// TIA Portal V19 export
DATA_BLOCK "DecoilersHRot"   // DB66
// stored: InstanceOfName DecoilersHRot_FB, InstanceOfType FB
"DecoilersHRot_FB"
   // VAR_INPUT
   //    AreaInterface : "AreaInterface";
   //    ZSI : "udt_ZoneSafetyInterface";
   //    DSI : Struct
   //       Rotation : "udt_DeviceSafetyInterface";
   //       Pivot : "udt_DeviceSafetyInterface";
   //       Translation : "udt_DeviceSafetyInterface";
   //    END_STRUCT;
   //    Drive : Struct
   //       Traslation : "TAx_DriveInterface";
   //    END_STRUCT;
   //    HW_ID : Struct
   //       Traslation_TEL1 : HW_SUBMODULE;
   //       TraslationEnc_IO : HW_SUBMODULE;
   //    END_STRUCT;
   //    DataIn : Struct
   //       PB_Decoiler1_MoveInLine : Bool;
   //       PB_Decoiler2_MoveInLine : Bool;
   //       Rotation : "ValveMachine_DataIn";
   //       Pivot : "ValveMachine_DataIn";
   //       Traslation : "Positioning_DOL_Machine_DataIn";
   //    END_STRUCT;
   //    CIn : Struct
   //       Manager : "DecoilersHRot_Manager";
   //       CoilCar_OutOfLine : Bool;
   //       PressureRunning_Rotation : Bool;
   //       PressureRunning_Pivot : Bool;
   //    END_STRUCT;
   //    Config : Struct
   //       Rotation : "ValveMachine_Config";
   //       Pivot : "ValveMachine_Config";
   //       Traslation : "Positioning_DOL_Machine_Config";
   //    END_STRUCT;
   // END_VAR
   // VAR_OUTPUT
   //    MachineInterface : "MachineInterface";
   //    DataOut : Struct
   //       Rotation : "ValveMachine_DataOut";
   //       Pivot : "ValveMachine_DataOut";
   //       Tower_Lamp : Bool;
   //       Tower_Horn : Bool;
   //    END_STRUCT;
   //    COut : "DecoilersHRot_Status";
   // END_VAR
   // VAR_IN_OUT
   //    PersistentValues : Struct
   //       Par : Struct
   //          TraslationAx : "Positioning_DOL_Machine_Par";
   //          TraslationEnc : "PosFbk_RTN";
   //          Traslation_AutSpeed : Real;
   //       END_STRUCT;
   //       Ax_Pers : "Positioning_DOL_Machine_Pers_Data";
   //    END_STRUCT;
   // END_VAR
   // VAR
   //    Warning : Struct
   //       Rotation : "ValveMachine_Wng";
   //       Pivot : "ValveMachine_Wng";
   //       Traslation : "Positioning_DOL_Machine_Wng";
   //       Rotation_NotInPosition : Bool;
   //       Pivot_NotWork : Bool;
   //       Translation_NotInPosition : Bool;
   //    END_STRUCT;
   //    Alarm : Struct
   //       Rotation : "ValveAlr";
   //       Pivot : "ValveAlr";
   //       Traslation_Ax : "Positioning_DOL_Machine_Alr";
   //       Traslation_Enc : "PosFbk_Encoder_Alr";
   //       Rotation_NotInPosition : Bool;
   //       Pivot_NotWork : Bool;
   //    END_STRUCT;
   //    Sts : Struct
   //       Decoiler1_InLine_Partial : Bool;
   //       Decoiler2_InLine_Partial : Bool;
   //    END_STRUCT;
   //    Ctrl : Struct
   //       Decoiler1_MoveInLine_Man : Bool;
   //       Decoiler2_MoveInLine_Man : Bool;
   //       Decoiler1_MoveInLine_Aut : Bool;
   //       Decoiler2_MoveInLine_Aut : Bool;
   //       Decoiler1_MoveInLine : Bool;
   //       Decoiler2_MoveInLine : Bool;
   //    END_STRUCT;
   //    Rotation : "ValveMachine_FB";
   //    Pivot : "ValveMachine_FB";
   //    Translation : "Positioning_DOL_Machine_FB";
   //    Traslation_Enc : "PosFbk_SickAFM60";
   //    Traslation_EncITF : "PosFbk_ITF";
   //    TON_Rotation_NotInPosition : TON_TIME;
   //    TON_Pivot_NotWork : TON_TIME;
   //    TON_Translation_NotInPosition { S7_SetPoint := 'True'} : TON_TIME;
   //    AUX : Struct
   //       Move_Pb_InLineDecoiler1 : Bool;
   //       Move_Pb_InLineDecoiler2 : Bool;
   //    END_STRUCT;
   // END_VAR
BEGIN
END_DATA_BLOCK
